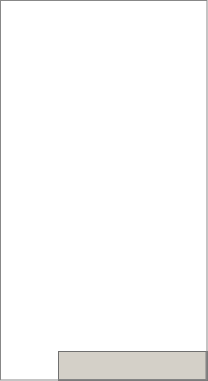
VISUALIZATION Visualization  // 208x381
    Button (58,351 150x30)
        tap Process.xStop
END_VISUALIZATION

(* stored: Version 1.1.0.1
   Visu Visualization: Id {123dee33-4147-47ad-9ee3-6f35a4bbe94b} *)
